// TIA Portal project "test" (V18)

(* hardware
DEVICE "ET 200SP station_1"  ET 200SP-Station
   slot 0: "Rack_0"  Rack  6ES5 710-8MAx1
   slot 1: "6ES7510-1DJ01-0AB0"  CPU 1510SP-1 PN  6ES7 510-1DJ01-0AB0  V2.9
      slot 32768: "PROFINET interface_1"  X1
         slot 32771: "Port_3"  X1 P3
   slot 3: "DI 16x24VDC ST_1"  DI 16x24VDC ST  6ES7 131-6BH01-0BA0  V0.0
      slot 1: "DI 16x24VDC ST_1"  DI 16x24VDC ST
   slot 4: "DQ 16x24VDC/0.5A ST_1"  DQ 16x24VDC/0.5A ST  6ES7 132-6BH01-0BA0  V0.0
      slot 1: "DQ 16x24VDC/0.5A ST_1"  DQ 16x24VDC/0.5A ST
   slot 5: "Server module_1"  Server module  6ES7 193-6PA00-0AA0  V1.1
      slot 1: "Server module_1"  Server module
   slot 127: "BA 2xRJ45"  BA 2xRJ45  6ES7 193-6AR00-0AA0  V0.0
      slot 32769: "Port_1"  X1 P1  6ES7 193-6AR00-0AA0
      slot 32770: "Port_2"  X1 P2  6ES7 193-6AR00-0AA0
   slot 33024: "DP interface_1"  CM DP Master/Slave  6ES7 545-5DA00-0AB0
DEVICE "ET 200S station_1"  ET 200S station
   slot 0: "Rack_0"  Rail
   slot 0: "Slave_1"  IM 151-1 Standard  6ES7 151-1AA06-0AB0  V4.0
   slot 1: "PM-E 24VDC_1"  PM-E 24VDC  6ES7 138-4CA01-0AA0
   slot 2: "8DI x 24VDC_1"  8DI x 24VDC  6ES7 131-4BF00-0AA0
   slot 3: "8DO x 24VDC / 0.5A_1"  8DO x 24VDC / 0.5A  6ES7 132-4BF00-0AA0
   slot 4: "2AO x U HS_1"  2AO x U HS  6ES7 135-4FB52-0AB0
   slot 5: "1 Count 24V_1"  1 COUNT 24V  6ES7 138-4DA04-0AB0  V2.0
*)

// ===== PLC "6ES7510-1DJ01-0AB0"  CPU 1510SP-1 PN =====

VAR_GLOBAL   // PLC tag table "Default tag table"
   "SB" AT %I0.0 : Bool;
   "HL" AT %Q0.0 : Bool;
   "Clock_Byte" AT %MB0 : Byte;
   "Clock_10Hz" AT %M0.0 : Bool;
   "Clock_5Hz" AT %M0.1 : Bool;
   "Clock_2.5Hz" AT %M0.2 : Bool;
   "Clock_2Hz" AT %M0.3 : Bool;
   "Clock_1.25Hz" AT %M0.4 : Bool;
   "Clock_1Hz" AT %M0.5 : Bool;
   "Clock_0.625Hz" AT %M0.6 : Bool;
   "Clock_0.5Hz" AT %M0.7 : Bool;
   "PROFIBUS_O" AT %Q2.0 : Bool;
   "COUNT" AT %ID8 : DInt;
   "SW_GATE" AT %Q12.0 : Bool;
   "ENGINE_CAPACITY" AT %QW4 : Int;
   "CONVERTER" AT %I2.0 : Bool;
END_VAR

DATA_BLOCK "CycleCheck_DB"   // DB1
{ S7_Optimized_Access := 'FALSE' }
VERSION : 0.1
// stored: InstanceOfName CycleCheck
"CycleCheck"
BEGIN
END_DATA_BLOCK

DATA_BLOCK "MyClock_DB"   // DB3
{ S7_Optimized_Access := 'FALSE' }
VERSION : 0.1
// stored: InstanceOfName MyClock
"MyClock"
BEGIN
END_DATA_BLOCK

FUNCTION_BLOCK "CycleCheck"   // FB1, SCL
{ S7_Optimized_Access := 'FALSE' }
VERSION : 0.1
   VAR
      temp : Bool;
      ie_value : DInt;
      last : DInt;
      flag : Bool;
      voltage : Real;
      temp_voltage : Int;
   END_VAR
BEGIN
   IF ("CONVERTER" OR "SB") AND NOT #temp THEN
       #temp := TRUE;
       "HL" := NOT "HL";
       "PROFIBUS_O" := NOT "PROFIBUS_O";
       "SW_GATE" := NOT "SW_GATE";
       #ie_value := 0;
   END_IF;

   IF NOT "SB" AND NOT "CONVERTER" THEN
       #temp := FALSE;
   END_IF;

   IF "SW_GATE" THEN
       IF #flag THEN
           IF #last < "COUNT" AND #ie_value > -1 AND #ie_value < 100 THEN
               #ie_value := #ie_value + 1;
           END_IF;
           IF #last > "COUNT" AND #ie_value > 0 AND #ie_value < 101 THEN
               #ie_value := #ie_value - 1;
           END_IF;
       ELSE
           IF "COUNT" > -1 AND "COUNT" < 101 THEN
               #ie_value := "COUNT";
           ELSE
               #flag := TRUE;
           END_IF;

       END_IF;
       #last := "COUNT";
   END_IF;

   #temp_voltage := REAL_TO_INT((DINT_TO_REAL(#ie_value) / 100.0) * 27648.0);

   IF #temp_voltage >= 0 AND #temp_voltage <= 27648 THEN
       "ENGINE_CAPACITY" := #temp_voltage;
       #voltage := DINT_TO_REAL(#ie_value) * 10.0;
   ELSE
       "ENGINE_CAPACITY" := 0;
       #voltage := 0.0;
   END_IF;

   "MyClock_DB"();
END_FUNCTION_BLOCK

FUNCTION_BLOCK "MyClock"   // FB2, SCL
{ S7_Optimized_Access := 'FALSE' }
VERSION : 0.1
   VAR
      seconds : Int;
      minutes : Int;
      hours : Int;
      temp : Bool;
   END_VAR
BEGIN
   IF "HL" THEN
       IF "Clock_0.5Hz" <> #temp THEN
           #temp := "Clock_0.5Hz";
           #seconds := #seconds + 1;
           IF #seconds = 60 THEN
               #seconds := 0;
               #minutes := #minutes + 1;
           END_IF;
           IF #minutes = 60 THEN
               #minutes := 0;
               #hours := #hours + 1;
           END_IF;
       END_IF;
   ELSE
       #seconds := 0;
       #minutes := 0;
       #hours := 0;
   END_IF;
END_FUNCTION_BLOCK

ORGANIZATION_BLOCK "Main"   // OB1, SCL, ProgramCycle
TITLE = "Main Program Sweep (Cycle)"
{ S7_Optimized_Access := 'TRUE' }
VERSION : 0.1
   VAR_INPUT
      Initial_Call : Bool;   // Initial call of this OB
      Remanence : Bool;   // =True, if remanent data are available
   END_VAR
BEGIN
   "CycleCheck_DB"();
END_ORGANIZATION_BLOCK